Omron CX-Programmer project NuevoProyecto (CX-Programmer 9.61)

# PLC NuevoPLC1: CQM1 CPU41

## Program NuevoPrograma1 (no task)
Local symbols
A_0 0.04 BOOL
A_1 0.05 BOOL
Am 100.04 BOOL
Amas 100.05 BOOL
B_0 0.07 BOOL
B_1 0.06 BOOL
Bm 100.07 BOOL
Bmas 100.06 BOOL
DI 0.09 BOOL
EM 17.03 BOOL
ET0 16.00 BOOL
ET1 16.01 BOOL
ET10 16.10 BOOL
ET11 16.11 BOOL
ET12 16.12 BOOL
ET13 16.13 BOOL
ET14 16.14 BOOL
ET15 16.15 BOOL
ET16 17.00 BOOL
ET2 16.02 BOOL
ET3 16.03 BOOL
ET4 16.04 BOOL
ET5 16.05 BOOL
ET6 16.06 BOOL
ET7 16.07 BOOL
ET8 16.08 BOOL
ET9 16.09 BOOL
F1 0.13 BOOL
F2 0.14 BOOL
FA 100.10 BOOL
FAUT 17.01 BOOL
FCI 0.08 BOOL
FCS 0.00 BOOL
FM 100.09 BOOL
FMAN 17.02 BOOL
KMB 100.08 BOOL
KMD 100.02 BOOL
KMI 100.01 BOOL
KMS 100.00 BOOL
LF1 100.13 BOOL
LF2 100.14 BOOL
LP 100.12 BOOL
LPA 100.15 BOOL
PINI 18.00 BOOL
PMB 0.10 BOOL
PMS 0.02 BOOL
PP 0.15 BOOL
SETC 100.03 BOOL
SMA 0.01 BOOL

### Section SET_RSET_ESTADOS

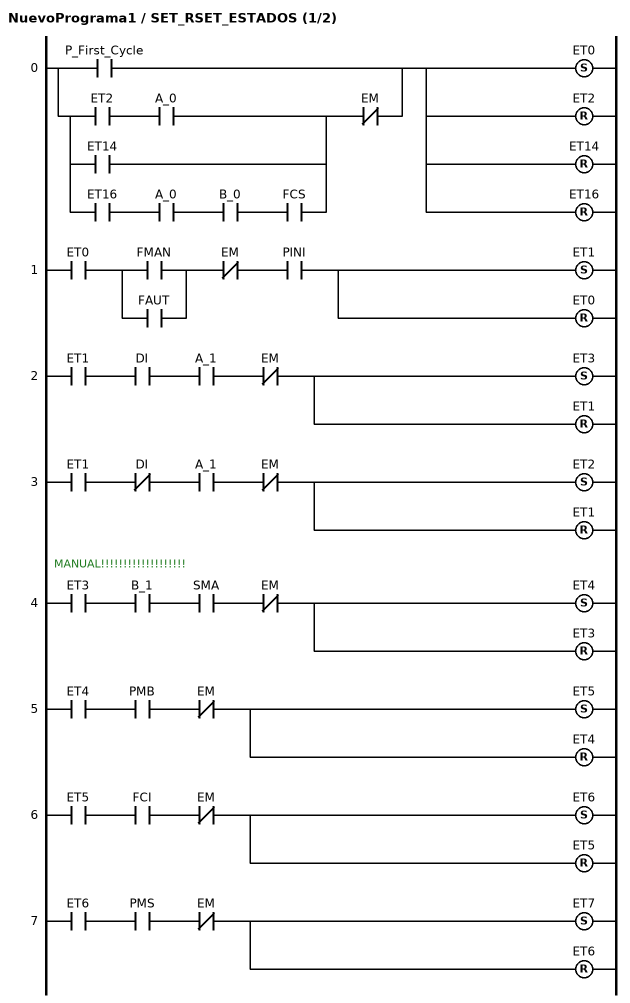
; rung 0
LD P_First_Cycle
LD ET2
AND A_0
OR ET14
LD ET16
AND A_0
AND B_0
AND FCS
ORLD
ANDNOT EM
ORLD
SET ET0
RSET ET2
RSET ET14
RSET ET16
; rung 1
LD ET0
LD FMAN
OR FAUT
ANDLD
ANDNOT EM
AND PINI
SET ET1
RSET ET0
; rung 2
LD ET1
AND DI
AND A_1
ANDNOT EM
SET ET3
RSET ET1
; rung 3
LD ET1
ANDNOT DI
AND A_1
ANDNOT EM
SET ET2
RSET ET1
; rung 4: MANUAL!!!!!!!!!!!!!!!!!!!
LD ET3
AND B_1
AND SMA
ANDNOT EM
SET ET4
RSET ET3
; rung 5
LD ET4
AND PMB
ANDNOT EM
SET ET5
RSET ET4
; rung 6
LD ET5
AND FCI
ANDNOT EM
SET ET6
RSET ET5
; rung 7
LD ET6
AND PMS
ANDNOT EM
SET ET7
RSET ET6

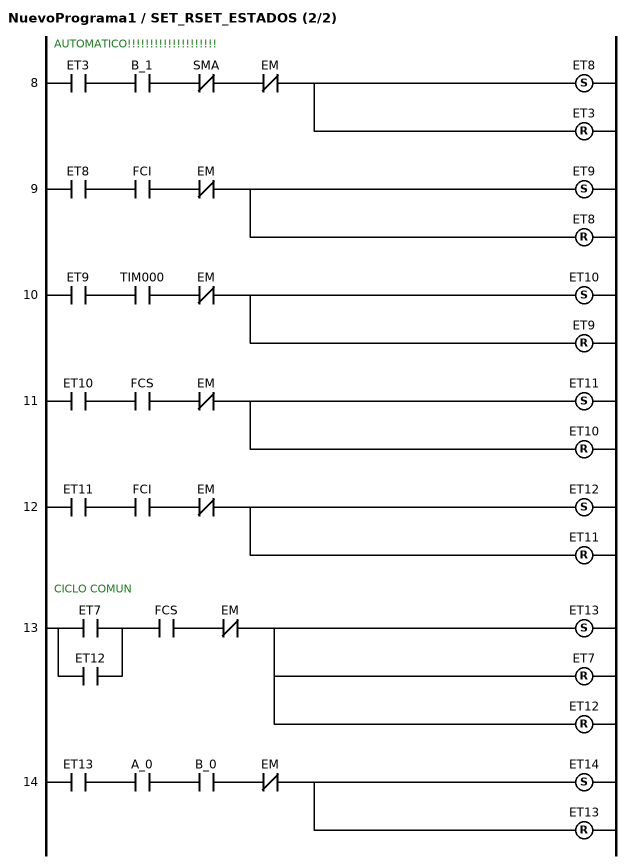
; rung 8: AUTOMATICO!!!!!!!!!!!!!!!!!!!!
LD ET3
AND B_1
ANDNOT SMA
ANDNOT EM
SET ET8
RSET ET3
; rung 9
LD ET8
AND FCI
ANDNOT EM
SET ET9
RSET ET8
; rung 10
LD ET9
AND TIM000
ANDNOT EM
SET ET10
RSET ET9
; rung 11
LD ET10
AND FCS
ANDNOT EM
SET ET11
RSET ET10
; rung 12
LD ET11
AND FCI
ANDNOT EM
SET ET12
RSET ET11
; rung 13: CICLO COMUN
LD ET7
OR ET12
AND FCS
ANDNOT EM
SET ET13
RSET ET7
RSET ET12
; rung 14
LD ET13
AND A_0
AND B_0
ANDNOT EM
SET ET14
RSET ET13

### Section ETAPAS

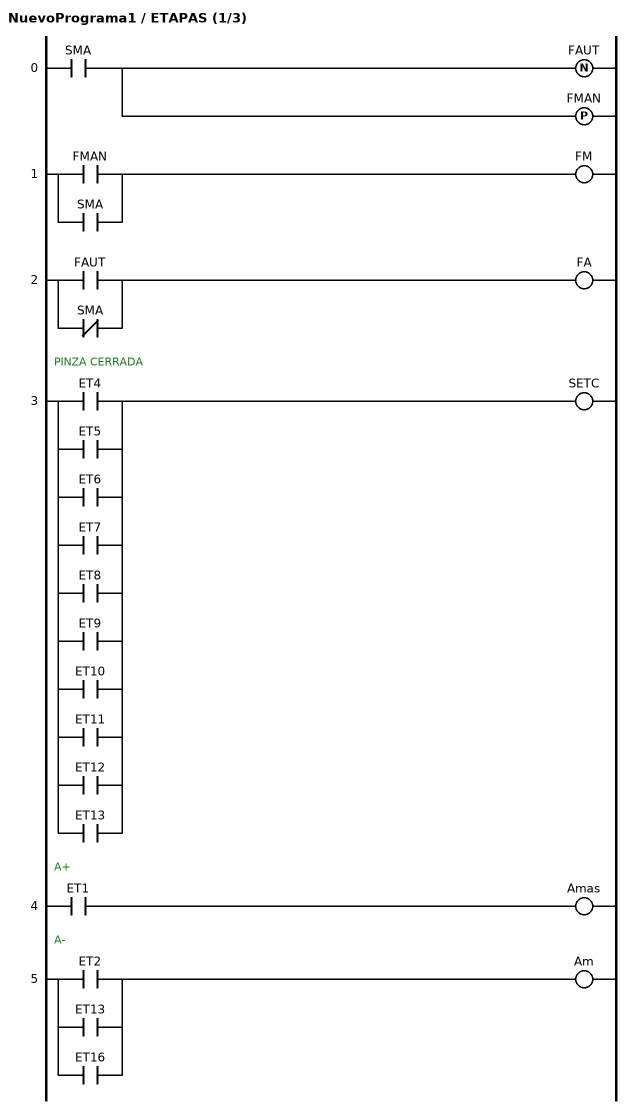
; rung 0
LD SMA
DIFD(14) FAUT
DIFU(13) FMAN
; rung 1
LD FMAN
OR SMA
OUT FM
; rung 2
LD FAUT
ORNOT SMA
OUT FA
; rung 3: PINZA CERRADA
LD ET4
OR ET5
OR ET6
OR ET7
OR ET8
OR ET9
OR ET10
OR ET11
OR ET12
OR ET13
OUT SETC
; rung 4: A+
LD ET1
OUT Amas
; rung 5: A-
LD ET2
OR ET13
OR ET16
OUT Am

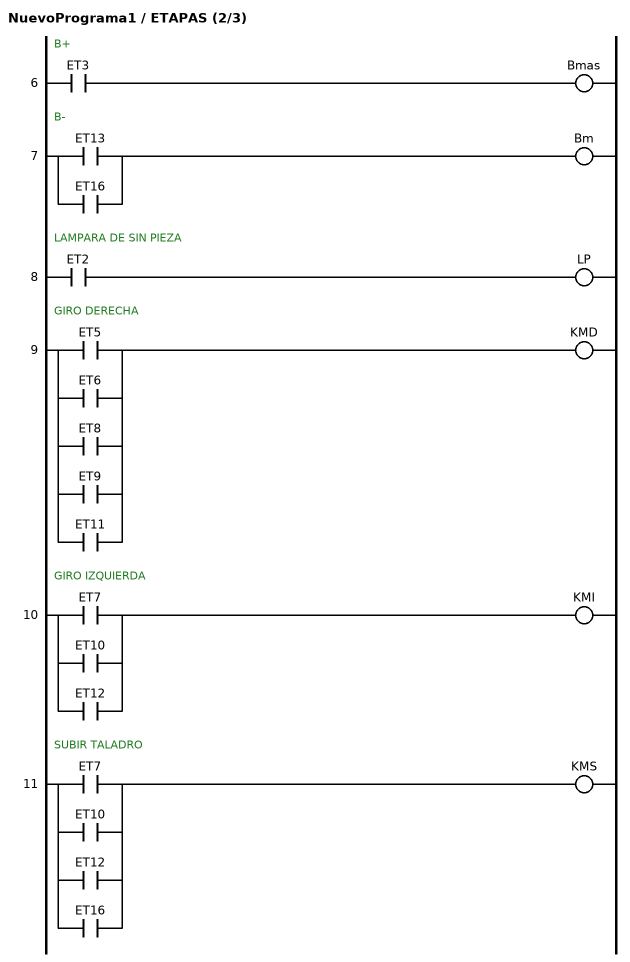
; rung 6: B+
LD ET3
OUT Bmas
; rung 7: B-
LD ET13
OR ET16
OUT Bm
; rung 8: LAMPARA DE SIN PIEZA
LD ET2
OUT LP
; rung 9: GIRO DERECHA
LD ET5
OR ET6
OR ET8
OR ET9
OR ET11
OUT KMD
; rung 10: GIRO IZQUIERDA
LD ET7
OR ET10
OR ET12
OUT KMI
; rung 11: SUBIR TALADRO
LD ET7
OR ET10
OR ET12
OR ET16
OUT KMS

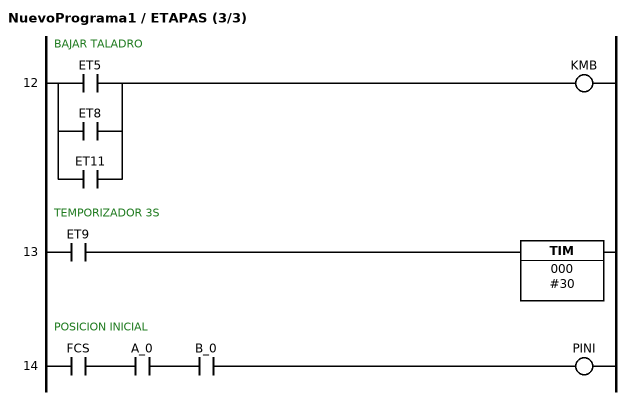
; rung 12: BAJAR TALADRO
LD ET5
OR ET8
OR ET11
OUT KMB
; rung 13: TEMPORIZADOR 3S
LD ET9
TIM 000 #30
; rung 14: POSICION INICIAL
LD FCS
AND A_0
AND B_0
OUT PINI

### Section EMERGENCIA

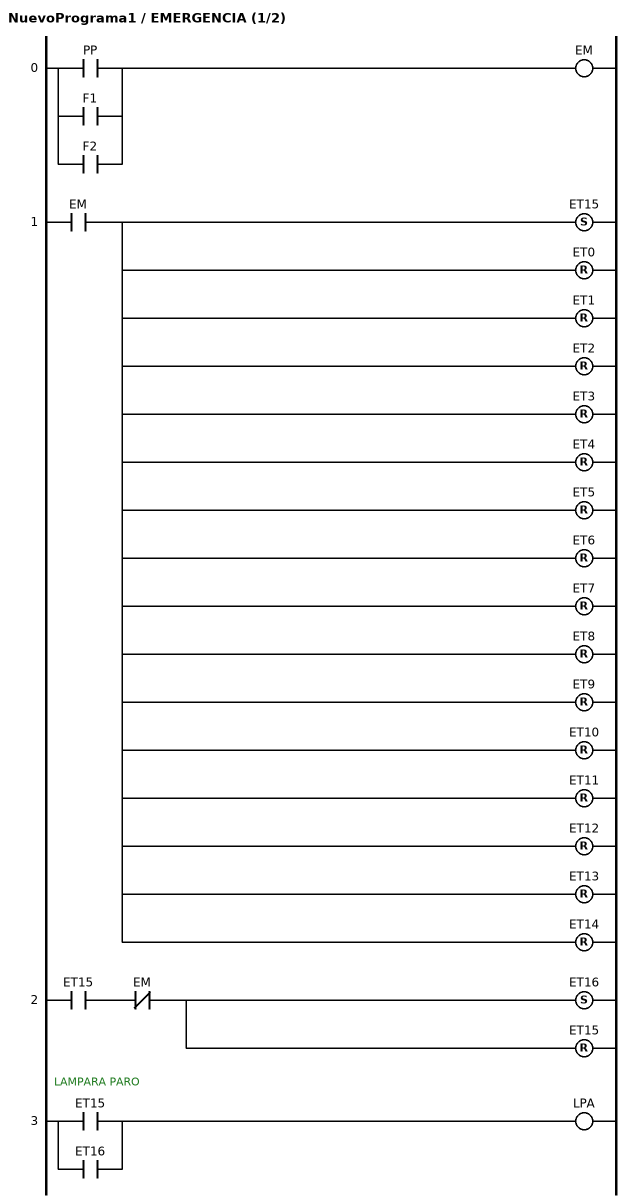
; rung 0
LD PP
OR F1
OR F2
OUT EM
; rung 1
LD EM
SET ET15
RSET ET0
RSET ET1
RSET ET2
RSET ET3
RSET ET4
RSET ET5
RSET ET6
RSET ET7
RSET ET8
RSET ET9
RSET ET10
RSET ET11
RSET ET12
RSET ET13
RSET ET14
; rung 2
LD ET15
ANDNOT EM
SET ET16
RSET ET15
; rung 3: LAMPARA PARO
LD ET15
OR ET16
OUT LPA

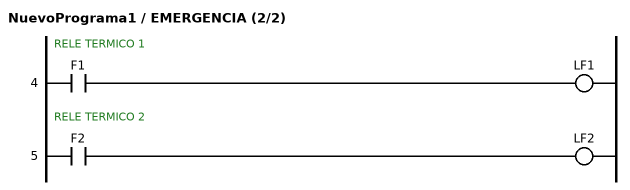
; rung 4: RELE TERMICO 1
LD F1
OUT LF1
; rung 5: RELE TERMICO 2
LD F2
OUT LF2

### Section END
; rung 0
END(01)